{attribute addProperty BoxType "EL3423-0000-0016"}
{attribute addProperty Id "Apparent_EnergyAT %I*LINT64818Apparent_Positive_EnergyAT %I*ULINT64819Apparent_Negative_EnergyAT %I*ULINT64820"}
{attribute addProperty CRC "2719322947"}
{attribute addProperty SizeInBites "192"}
{attribute addProperty SizeInBytes "24"}
TYPE Total_Apparent_A2159343 :
STRUCT
	{attribute addProperty Name "Apparent_Energy"}
	Apparent_Energy AT %I* : LINT;
	{attribute addProperty Name "Apparent_Positive_Energy"}
	Apparent_Positive_Energy AT %I* : ULINT;
	{attribute addProperty Name "Apparent_Negative_Energy"}
	Apparent_Negative_Energy AT %I* : ULINT;
END_STRUCT
END_TYPE

(* stored: Version 1.2.0.0, ProductVersion 3.1.4024.9
   DUT Total_Apparent_A2159343: Id {6b3c47b3-a8b7-4f1c-b6fd-598dee0c5b25} *)
